TYPE st_InfoDataGroup :
STRUCT
	state,diag:USINT;
END_STRUCT
END_TYPE

(* stored: Version 1.1.0.1, ProductVersion 3.1.4024.12
   DUT st_InfoDataGroup: Id {39566151-30da-4901-945c-44195fbfffa8} *)
